{attribute 'qualified_only'}
{attribute 'strict'}
{attribute 'to_string'}
TYPE E_FilterType :
(
    None := 0,
    FixedThickness,
    Wedge
);
END_TYPE

(* stored: Version 1.1.0.1
   DUT E_FilterType: Id {64eb8815-a5b7-4702-a855-ca6a3bc89090} *)
